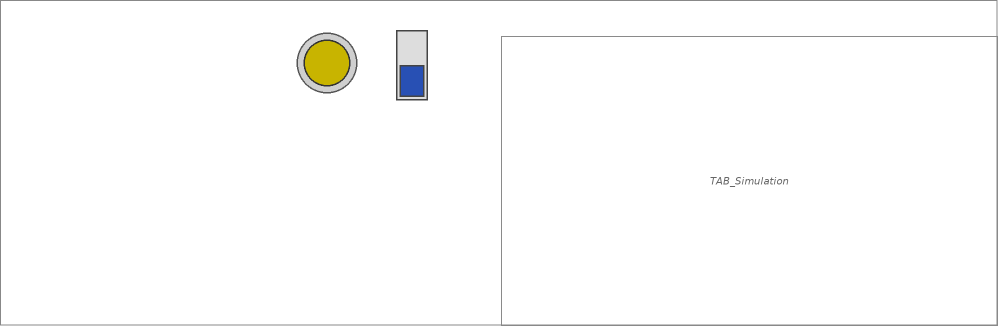
VISUALIZATION HMI  // 998x326
    TabControl (501,36 497x290)
        shows TAB_Simulation()
    DipSwitch (377,30 70x70), variable: Temp.bSwitch1, behaviour: TOGGLE, style: Switch-DipSwitch-Blue
    Lamp1 (292,28 70x70), variable: Temp.bLED1, style: Lamp-Lamp1-Yellow
END_VISUALIZATION

(* stored: Version 1.1.0.1, ProductVersion 3.1.4024.11
   Visu HMI: Id {e83fe0f6-a3fa-41e5-916a-5fed390733ae} *)
